(* CoDeSys 2.3 export: PHYSICAL.EXP *)

(* Global variable list: physical *)
VAR_GLOBAL
	din1_1	AT %IX52.0:	BOOL;
	din1_2	AT %IX52.1:	BOOL;
	din1_3	AT %IX52.2:	BOOL;
	din1_4	AT %IX52.3:	BOOL;
	din1_5	AT %IX52.4:	BOOL;
	din1_6	AT %IX52.5:	BOOL;
	din1_7	AT %IX52.6:	BOOL;
	din1_8	AT %IX52.7:	BOOL;
	din2_1	AT %IX53.0:	BOOL;
	din2_2	AT %IX53.1:	BOOL;
	din2_3	AT %IX53.2:	BOOL;
	din2_4	AT %IX53.3:	BOOL;
	din2_5	AT %IX53.4:	BOOL;
	din2_6	AT %IX53.5:	BOOL;
	din2_7	AT %IX53.6:	BOOL;
	din2_8	AT %IX53.7:	BOOL;
(*din3_1*)sw_kino_balkon	AT %IX54.0:	BOOL;
(*din3_2*)sw_tambur2		AT %IX54.1:	BOOL;
(*din3_3*)sw_kino1			AT %IX54.2:	BOOL;
(*din3_4*)sw_korydor		AT %IX54.3:	BOOL;
(*din3_5*)sw_kino2			AT %IX54.4:	BOOL;
(*din3_6*)sw_studio1			AT %IX54.5:	BOOL;
(*din3_7*)sw_tambur1		AT %IX54.6:	BOOL;
(*din3_8*)sw_studio2			AT %IX54.7:	BOOL;
(*din4_1*)sw_kabinet1		AT %IX55.0:	BOOL;
	din4_2	AT %IX55.1:	BOOL;
(*din4_3*)sw_kabinet2	AT %IX55.2:	BOOL;
(*din4_4*)sw_kabinet2_1	AT %IX55.3:	BOOL;
(*din4_5*)sw_kabinet_balkon	AT %IX55.4:	BOOL;
(*din4_6*)sw_kabinet2_2	AT %IX55.5:	BOOL;
(*din4_7*)sw_tambur3		AT %IX55.6:	BOOL;
	din4_8	AT %IX55.7:	BOOL;

(*dout1_1*)balkon_peryla				AT %QX52.0:	BOOL;
(*dout1_2*)kino_l					AT %QX52.1:	BOOL;
(*dout1_3*)balkon_bra				AT %QX52.2:	BOOL;
(*dout1_4*)kabinet_balkon_l			AT %QX52.3:	BOOL;
(*dout1_5*)balkon					AT %QX52.4:	BOOL;
(*dout1_6*)korydor1					AT %QX52.5:	BOOL;
(*dout1_7*)kino_bra					AT %QX52.6:	BOOL;
(*dout1_8*)korydor2					AT %QX52.7:	BOOL;
(*dout2_1*)studio_pidsvitka 			AT %QX53.0:	BOOL;
(*dout2_2*)skhody2_3				AT %QX53.1:	BOOL;
(*dout2_3*)studio_l					AT %QX53.2:	BOOL;
(*dout2_4*)kabinet_pidsvitka_kolo	AT %QX53.3:	BOOL;
(*dout2_5*)kabinet_svitlo				AT %QX53.4:	BOOL;
(*dout2_6*)kabinet_kobra 			AT %QX53.5:	BOOL;
(*dout2_7*)tambur_l					AT %QX53.6:	BOOL;
	stend	AT %QX53.7:	BOOL;
(*dout3_1*)collector_kabinet1		AT %QX54.0:	BOOL;
(*dout3_2*)fancoil_kabinet_low		AT %QX54.1:	BOOL;
(*dout3_3*)collector_kabinet2		AT %QX54.2:	BOOL;
(*dout3_4*)fancoil_kabinet_med		AT %QX54.3:	BOOL;
(*dout3_5*)collector_studio1			AT %QX54.4:	BOOL;
	fancoil_kabinet_high				AT %QX54.5:	BOOL;
(*dout3_7*)collector_studio2			AT %QX54.6:	BOOL;
(*dout3_8*)fancoil_kino_low			AT %QX54.7:	BOOL;
(*dout4_1*)fancoil_kino_med		AT %QX55.0:	BOOL;
	dout4_2	AT %QX55.1:	BOOL;
	fancoil_kino_high				AT %QX55.2:	BOOL;
	skhody_peryla	AT %QX55.3:	BOOL;
	dout4_5	AT %QX55.4:	BOOL;
	dout4_6	AT %QX55.5:	BOOL;
	dout4_7	AT %QX55.6:	BOOL;
	dout4_8	AT %QX55.7:	BOOL;
	kino_tul_open			AT %QX56.0:	BOOL;
	kabinet_tul_open 		AT %QX56.1:	BOOL;
	kino_tul_close 			AT %QX56.2:	BOOL;
	kabinet_tul_close		AT %QX56.3:	BOOL;
	kino_shtory_open		AT %QX56.4:	BOOL;
	kabinet_shtory_open	AT %QX56.5:	BOOL;
	kino_shtory_close		AT %QX56.6:	BOOL;
	kabinet_shtory_close	AT %QX56.7:	BOOL;


	klapan_kino 	AT %QB2:	INT;
	klapan_kabinet	AT %QB6:	INT;
	test1 AT %IB51:BYTE;
	test2 AT %IB2:BYTE;
	test3 AT %IB10:BYTE;
	test4 AT %IB54:BYTE;
	test5 AT %IB55:BYTE;
	test6 AT %IB56:BYTE;
	test7 AT %IB57:BYTE;
	test8 AT %IB58:BYTE;
	test9 AT %IB59:BYTE;
	test10 AT %IB60:BYTE;
	test11 AT %IB61:BYTE;
	test12 AT %IB62:BYTE;
	test13 AT %IB63:BYTE;
	test14 AT %IB64:BYTE;
	test15 AT %IB65:BYTE;

	Term_2_KL4414_1_State	AT %IB0:	USINT;
	Term_2_KL4414_1_Data_In	AT %IB2:	INT;
	Term_2_KL4414_1_Ctrl	AT %QB0:	USINT;
	Term_2_KL4414_1_Data_Out	AT %QB2:	INT;
	Term_2_KL4414_2_State	AT %IB4:	USINT;
	Term_2_KL4414_2_Data_In	AT %IB6:	INT;
	Term_2_KL4414_2_Ctrl	AT %QB4:	USINT;
	Term_2_KL4414_2_Data_Out	AT %QB6:	INT;
	Term_2_KL4414_3_State	AT %IB8:	USINT;
	Term_2_KL4414_3_Data_In	AT %IB10:	INT;
	Term_2_KL4414_3_Ctrl	AT %QB8:	USINT;
	Term_2_KL4414_3_Data_Out	AT %QB10:	INT;
	Term_2_KL4414_4_State	AT %IB12:	USINT;
	Term_2_KL4414_4_Data_In	AT %IB14:	INT;
	Term_2_KL4414_4_Ctrl	AT %QB12:	USINT;
	Term_2_KL4414_4_Data_Out	AT %QB14:	INT;
	Term_12_KL3228_4_1_State	AT %IB16:	USINT;
	Term_12_KL3228_4_1_Data_In	AT %IB18:	INT;
	Term_12_KL3228_4_1_Ctrl	AT %QB16:	USINT;
	Term_12_KL3228_4_1_Data_Out	AT %QB18:	INT;
	Term_12_KL3228_4_2_State	AT %IB20:	USINT;
	Term_12_KL3228_4_2_Data_In	AT %IB22:	INT;
	Term_12_KL3228_4_2_Ctrl	AT %QB20:	USINT;
	Term_12_KL3228_4_2_Data_Out	AT %QB22:	INT;
	Term_12_KL3228_4_3_State	AT %IB24:	USINT;
	Term_12_KL3228_4_3_Data_In	AT %IB26:	INT;
	Term_12_KL3228_4_3_Ctrl	AT %QB24:	USINT;
	Term_12_KL3228_4_3_Data_Out	AT %QB26:	INT;
	Term_12_KL3228_4_4_State	AT %IB28:	USINT;
	Term_12_KL3228_4_4_Data_In	AT %IB30:	INT;
	Term_12_KL3228_4_4_Ctrl	AT %QB28:	USINT;
	Term_12_KL3228_4_4_Data_Out	AT %QB30:	INT;
	Term_13_KL3228_4_1_State	AT %IB32:	USINT;
	Term_13_KL3228_4_1_Data_In	AT %IB34:	INT;
	Term_13_KL3228_4_1_Ctrl	AT %QB32:	USINT;
	Term_13_KL3228_4_1_Data_Out	AT %QB34:	INT;
	Term_13_KL3228_4_2_State	AT %IB36:	USINT;
	Term_13_KL3228_4_2_Data_In	AT %IB38:	INT;
	Term_13_KL3228_4_2_Ctrl	AT %QB36:	USINT;
	Term_13_KL3228_4_2_Data_Out	AT %QB38:	INT;
	Term_13_KL3228_4_3_State	AT %IB40:	USINT;
	Term_13_KL3228_4_3_Data_In	AT %IB42:	INT;
	Term_13_KL3228_4_3_Ctrl	AT %QB40:	USINT;
	Term_13_KL3228_4_3_Data_Out	AT %QB42:	INT;
	Term_13_KL3228_4_4_State	AT %IB44:	USINT;
	Term_13_KL3228_4_4_Data_In	AT %IB46:	INT;
	Term_13_KL3228_4_4_Ctrl	AT %QB44:	USINT;
	Term_13_KL3228_4_4_Data_Out	AT %QB46:	INT;
	Term_14_KL2761_State	AT %IB48:	USINT;
	Term_14_KL2761_Data_In	AT %IB50:	INT;
	Term_14_KL2761_Ctrl	AT %QB48:	USINT;
	Term_14_KL2761_Data_Out	AT %QB50:	INT;
	(*Term_2_KL3228_4_1_Data_In	AT %IB2:	INT; (*-45*)
	Term_2_KL3228_4_3_Data_In	AT %IB10:	INT; (*-45*)
*)


END_VAR
(*
